// TIA Portal V17 export
// export: Created 2026-04-12T10:31:24.245585Z, ExportSetting WithDefaults, DisplayName Totally Integrated Automation Portal, DisplayVersion V17 Update 4, DisplayName TIA Portal Openness, DisplayVersion V17 Update 4, DisplayName TIA Portal Version Control Interface, DisplayVersion V17, DisplayName SINAMICS Startdrive Advanced, DisplayVersion V17, DisplayName SINAMICS Startdrive G130, G150, S120, S150, SINAMICS MV, S210, DisplayVersion V17, DisplayName SINAMICS Startdrive G110M, G120, G120C, G120D, G120P, G115D, DisplayVersion V17, DisplayName STEP 7 Professional, DisplayVersion V17 Update 4, DisplayName STEP 7 Safety, DisplayVersion V17, DisplayName WinCC Advanced, DisplayVersion V17 Update 4
FUNCTION "烧嘴控制块" : Void   // FC4, LAD
{ S7_Optimized_Access := 'TRUE' }
VERSION : 0.1
// stored: AutoNumber true, IsIECCheckEnabled false, SetENOAutomatically false, UDAEnableTagReadback false
   VAR_TEMP   // added for the SCL form of the ladder/FBD networks
      _w1 : Bool;
      _w2 : Bool;
   END_VAR
BEGIN

REGION Network 1: 1#烧嘴控制
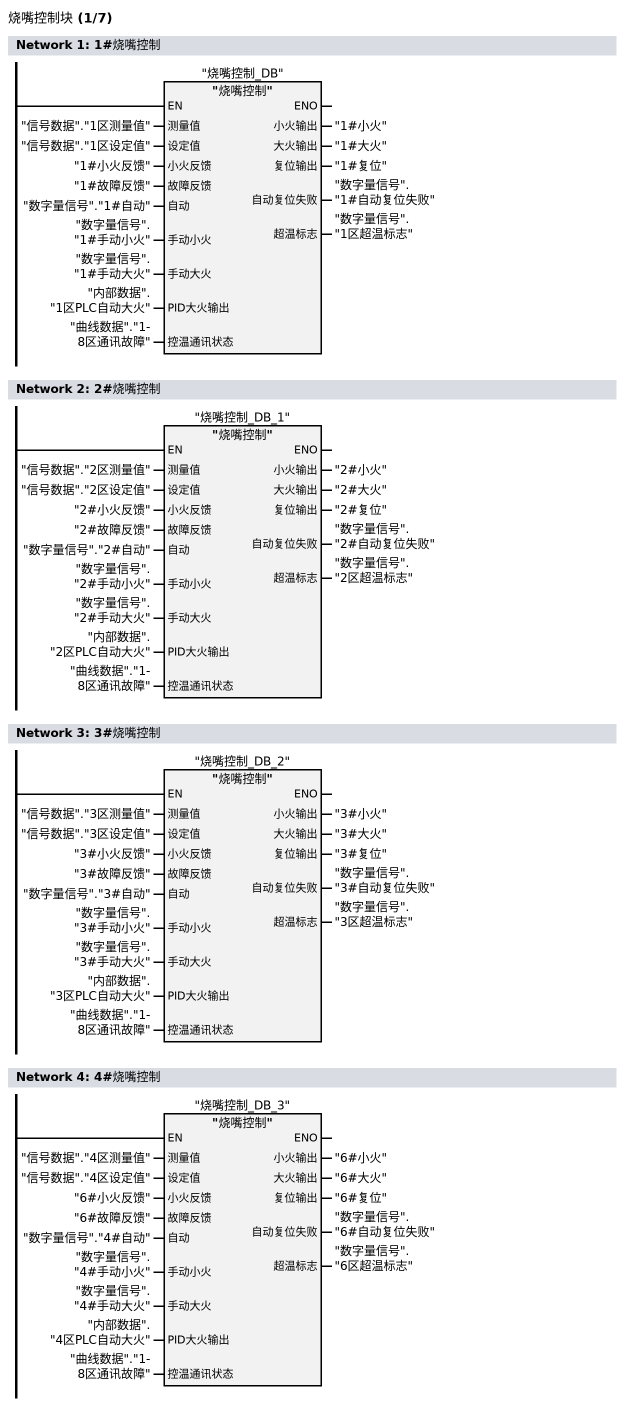
   RUNG wire#powerrail
      "烧嘴控制_DB"(测量值 := "信号数据"."1区测量值", 设定值 := "信号数据"."1区设定值", 小火反馈 := "1#小火反馈", 故障反馈 := "1#故障反馈", 自动 := "数字量信号"."1#自动", 手动小火 := "数字量信号"."1#手动小火", 手动大火 := "数字量信号"."1#手动大火", PID大火输出 := "内部数据"."1区PLC自动大火", 控温通讯状态 := "曲线数据"."1-8区通讯故障", 小火输出 => "1#小火", 大火输出 => "1#大火", 复位输出 => "1#复位", 自动复位失败 => "数字量信号"."1#自动复位失败", 超温标志 => "数字量信号"."1区超温标志")
   END_RUNG
   // the same network as SCL:
   "烧嘴控制_DB"(测量值 := "信号数据"."1区测量值",   // "烧嘴控制"
             设定值 := "信号数据"."1区设定值",
             小火反馈 := "1#小火反馈",
             故障反馈 := "1#故障反馈",
             自动 := "数字量信号"."1#自动",
             手动小火 := "数字量信号"."1#手动小火",
             手动大火 := "数字量信号"."1#手动大火",
             PID大火输出 := "内部数据"."1区PLC自动大火",
             控温通讯状态 := "曲线数据"."1-8区通讯故障",
             小火输出 => "1#小火",
             大火输出 => "1#大火",
             复位输出 => "1#复位",
             自动复位失败 => "数字量信号"."1#自动复位失败",
             超温标志 => "数字量信号"."1区超温标志");
END_REGION

REGION Network 2: 2#烧嘴控制
   RUNG wire#powerrail
      "烧嘴控制_DB_1"(测量值 := "信号数据"."2区测量值", 设定值 := "信号数据"."2区设定值", 小火反馈 := "2#小火反馈", 故障反馈 := "2#故障反馈", 自动 := "数字量信号"."2#自动", 手动小火 := "数字量信号"."2#手动小火", 手动大火 := "数字量信号"."2#手动大火", PID大火输出 := "内部数据"."2区PLC自动大火", 控温通讯状态 := "曲线数据"."1-8区通讯故障", 小火输出 => "2#小火", 大火输出 => "2#大火", 复位输出 => "2#复位", 自动复位失败 => "数字量信号"."2#自动复位失败", 超温标志 => "数字量信号"."2区超温标志")
   END_RUNG
   // the same network as SCL:
   "烧嘴控制_DB_1"(测量值 := "信号数据"."2区测量值",   // "烧嘴控制"
               设定值 := "信号数据"."2区设定值",
               小火反馈 := "2#小火反馈",
               故障反馈 := "2#故障反馈",
               自动 := "数字量信号"."2#自动",
               手动小火 := "数字量信号"."2#手动小火",
               手动大火 := "数字量信号"."2#手动大火",
               PID大火输出 := "内部数据"."2区PLC自动大火",
               控温通讯状态 := "曲线数据"."1-8区通讯故障",
               小火输出 => "2#小火",
               大火输出 => "2#大火",
               复位输出 => "2#复位",
               自动复位失败 => "数字量信号"."2#自动复位失败",
               超温标志 => "数字量信号"."2区超温标志");
END_REGION

REGION Network 3: 3#烧嘴控制
   RUNG wire#powerrail
      "烧嘴控制_DB_2"(测量值 := "信号数据"."3区测量值", 设定值 := "信号数据"."3区设定值", 小火反馈 := "3#小火反馈", 故障反馈 := "3#故障反馈", 自动 := "数字量信号"."3#自动", 手动小火 := "数字量信号"."3#手动小火", 手动大火 := "数字量信号"."3#手动大火", PID大火输出 := "内部数据"."3区PLC自动大火", 控温通讯状态 := "曲线数据"."1-8区通讯故障", 小火输出 => "3#小火", 大火输出 => "3#大火", 复位输出 => "3#复位", 自动复位失败 => "数字量信号"."3#自动复位失败", 超温标志 => "数字量信号"."3区超温标志")
   END_RUNG
   // the same network as SCL:
   "烧嘴控制_DB_2"(测量值 := "信号数据"."3区测量值",   // "烧嘴控制"
               设定值 := "信号数据"."3区设定值",
               小火反馈 := "3#小火反馈",
               故障反馈 := "3#故障反馈",
               自动 := "数字量信号"."3#自动",
               手动小火 := "数字量信号"."3#手动小火",
               手动大火 := "数字量信号"."3#手动大火",
               PID大火输出 := "内部数据"."3区PLC自动大火",
               控温通讯状态 := "曲线数据"."1-8区通讯故障",
               小火输出 => "3#小火",
               大火输出 => "3#大火",
               复位输出 => "3#复位",
               自动复位失败 => "数字量信号"."3#自动复位失败",
               超温标志 => "数字量信号"."3区超温标志");
END_REGION

REGION Network 4: 4#烧嘴控制
   RUNG wire#powerrail
      "烧嘴控制_DB_3"(测量值 := "信号数据"."4区测量值", 设定值 := "信号数据"."4区设定值", 小火反馈 := "6#小火反馈", 故障反馈 := "6#故障反馈", 自动 := "数字量信号"."4#自动", 手动小火 := "数字量信号"."4#手动小火", 手动大火 := "数字量信号"."4#手动大火", PID大火输出 := "内部数据"."4区PLC自动大火", 控温通讯状态 := "曲线数据"."1-8区通讯故障", 小火输出 => "6#小火", 大火输出 => "6#大火", 复位输出 => "6#复位", 自动复位失败 => "数字量信号"."6#自动复位失败", 超温标志 => "数字量信号"."6区超温标志")
   END_RUNG
   // the same network as SCL:
   "烧嘴控制_DB_3"(测量值 := "信号数据"."4区测量值",   // "烧嘴控制"
               设定值 := "信号数据"."4区设定值",
               小火反馈 := "6#小火反馈",
               故障反馈 := "6#故障反馈",
               自动 := "数字量信号"."4#自动",
               手动小火 := "数字量信号"."4#手动小火",
               手动大火 := "数字量信号"."4#手动大火",
               PID大火输出 := "内部数据"."4区PLC自动大火",
               控温通讯状态 := "曲线数据"."1-8区通讯故障",
               小火输出 => "6#小火",
               大火输出 => "6#大火",
               复位输出 => "6#复位",
               自动复位失败 => "数字量信号"."6#自动复位失败",
               超温标志 => "数字量信号"."6区超温标志");
END_REGION

REGION Network 5: 5#烧嘴控制
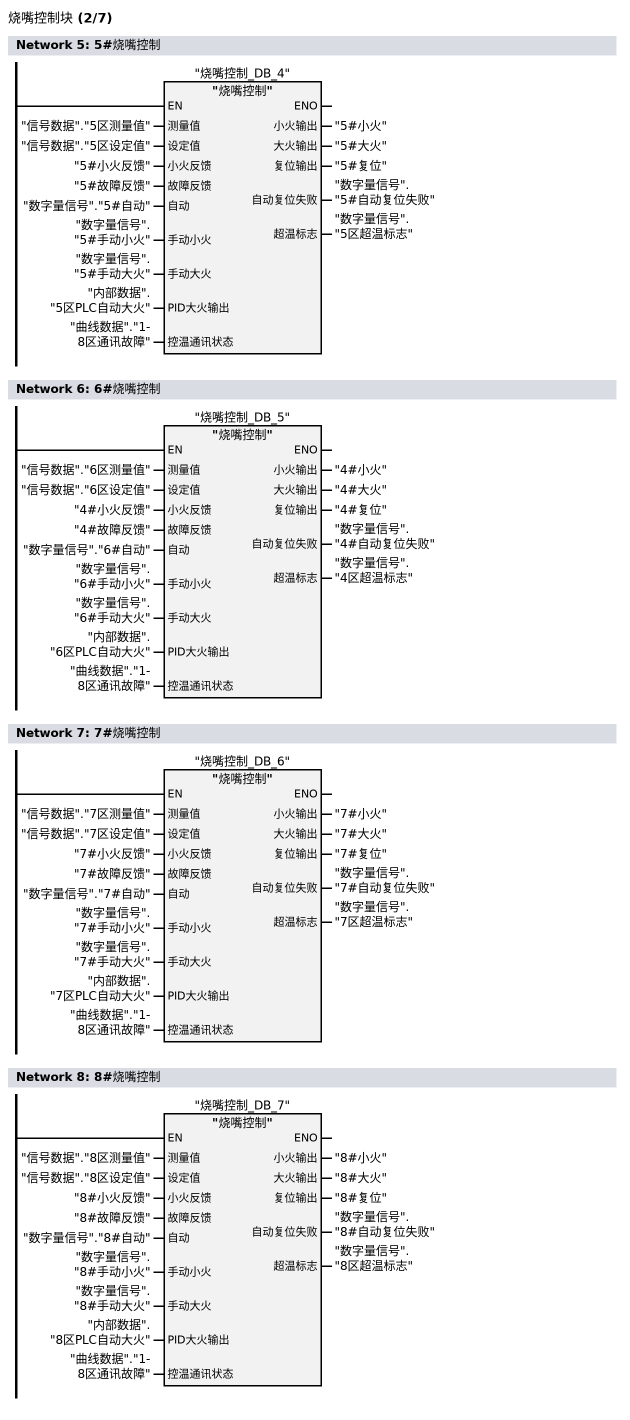
   RUNG wire#powerrail
      "烧嘴控制_DB_4"(测量值 := "信号数据"."5区测量值", 设定值 := "信号数据"."5区设定值", 小火反馈 := "5#小火反馈", 故障反馈 := "5#故障反馈", 自动 := "数字量信号"."5#自动", 手动小火 := "数字量信号"."5#手动小火", 手动大火 := "数字量信号"."5#手动大火", PID大火输出 := "内部数据"."5区PLC自动大火", 控温通讯状态 := "曲线数据"."1-8区通讯故障", 小火输出 => "5#小火", 大火输出 => "5#大火", 复位输出 => "5#复位", 自动复位失败 => "数字量信号"."5#自动复位失败", 超温标志 => "数字量信号"."5区超温标志")
   END_RUNG
   // the same network as SCL:
   "烧嘴控制_DB_4"(测量值 := "信号数据"."5区测量值",   // "烧嘴控制"
               设定值 := "信号数据"."5区设定值",
               小火反馈 := "5#小火反馈",
               故障反馈 := "5#故障反馈",
               自动 := "数字量信号"."5#自动",
               手动小火 := "数字量信号"."5#手动小火",
               手动大火 := "数字量信号"."5#手动大火",
               PID大火输出 := "内部数据"."5区PLC自动大火",
               控温通讯状态 := "曲线数据"."1-8区通讯故障",
               小火输出 => "5#小火",
               大火输出 => "5#大火",
               复位输出 => "5#复位",
               自动复位失败 => "数字量信号"."5#自动复位失败",
               超温标志 => "数字量信号"."5区超温标志");
END_REGION

REGION Network 6: 6#烧嘴控制
   RUNG wire#powerrail
      "烧嘴控制_DB_5"(测量值 := "信号数据"."6区测量值", 设定值 := "信号数据"."6区设定值", 小火反馈 := "4#小火反馈", 故障反馈 := "4#故障反馈", 自动 := "数字量信号"."6#自动", 手动小火 := "数字量信号"."6#手动小火", 手动大火 := "数字量信号"."6#手动大火", PID大火输出 := "内部数据"."6区PLC自动大火", 控温通讯状态 := "曲线数据"."1-8区通讯故障", 小火输出 => "4#小火", 大火输出 => "4#大火", 复位输出 => "4#复位", 自动复位失败 => "数字量信号"."4#自动复位失败", 超温标志 => "数字量信号"."4区超温标志")
   END_RUNG
   // the same network as SCL:
   "烧嘴控制_DB_5"(测量值 := "信号数据"."6区测量值",   // "烧嘴控制"
               设定值 := "信号数据"."6区设定值",
               小火反馈 := "4#小火反馈",
               故障反馈 := "4#故障反馈",
               自动 := "数字量信号"."6#自动",
               手动小火 := "数字量信号"."6#手动小火",
               手动大火 := "数字量信号"."6#手动大火",
               PID大火输出 := "内部数据"."6区PLC自动大火",
               控温通讯状态 := "曲线数据"."1-8区通讯故障",
               小火输出 => "4#小火",
               大火输出 => "4#大火",
               复位输出 => "4#复位",
               自动复位失败 => "数字量信号"."4#自动复位失败",
               超温标志 => "数字量信号"."4区超温标志");
END_REGION

REGION Network 7: 7#烧嘴控制
   RUNG wire#powerrail
      "烧嘴控制_DB_6"(测量值 := "信号数据"."7区测量值", 设定值 := "信号数据"."7区设定值", 小火反馈 := "7#小火反馈", 故障反馈 := "7#故障反馈", 自动 := "数字量信号"."7#自动", 手动小火 := "数字量信号"."7#手动小火", 手动大火 := "数字量信号"."7#手动大火", PID大火输出 := "内部数据"."7区PLC自动大火", 控温通讯状态 := "曲线数据"."1-8区通讯故障", 小火输出 => "7#小火", 大火输出 => "7#大火", 复位输出 => "7#复位", 自动复位失败 => "数字量信号"."7#自动复位失败", 超温标志 => "数字量信号"."7区超温标志")
   END_RUNG
   // the same network as SCL:
   "烧嘴控制_DB_6"(测量值 := "信号数据"."7区测量值",   // "烧嘴控制"
               设定值 := "信号数据"."7区设定值",
               小火反馈 := "7#小火反馈",
               故障反馈 := "7#故障反馈",
               自动 := "数字量信号"."7#自动",
               手动小火 := "数字量信号"."7#手动小火",
               手动大火 := "数字量信号"."7#手动大火",
               PID大火输出 := "内部数据"."7区PLC自动大火",
               控温通讯状态 := "曲线数据"."1-8区通讯故障",
               小火输出 => "7#小火",
               大火输出 => "7#大火",
               复位输出 => "7#复位",
               自动复位失败 => "数字量信号"."7#自动复位失败",
               超温标志 => "数字量信号"."7区超温标志");
END_REGION

REGION Network 8: 8#烧嘴控制
   RUNG wire#powerrail
      "烧嘴控制_DB_7"(测量值 := "信号数据"."8区测量值", 设定值 := "信号数据"."8区设定值", 小火反馈 := "8#小火反馈", 故障反馈 := "8#故障反馈", 自动 := "数字量信号"."8#自动", 手动小火 := "数字量信号"."8#手动小火", 手动大火 := "数字量信号"."8#手动大火", PID大火输出 := "内部数据"."8区PLC自动大火", 控温通讯状态 := "曲线数据"."1-8区通讯故障", 小火输出 => "8#小火", 大火输出 => "8#大火", 复位输出 => "8#复位", 自动复位失败 => "数字量信号"."8#自动复位失败", 超温标志 => "数字量信号"."8区超温标志")
   END_RUNG
   // the same network as SCL:
   "烧嘴控制_DB_7"(测量值 := "信号数据"."8区测量值",   // "烧嘴控制"
               设定值 := "信号数据"."8区设定值",
               小火反馈 := "8#小火反馈",
               故障反馈 := "8#故障反馈",
               自动 := "数字量信号"."8#自动",
               手动小火 := "数字量信号"."8#手动小火",
               手动大火 := "数字量信号"."8#手动大火",
               PID大火输出 := "内部数据"."8区PLC自动大火",
               控温通讯状态 := "曲线数据"."1-8区通讯故障",
               小火输出 => "8#小火",
               大火输出 => "8#大火",
               复位输出 => "8#复位",
               自动复位失败 => "数字量信号"."8#自动复位失败",
               超温标志 => "数字量信号"."8区超温标志");
END_REGION

REGION Network 9: 9#烧嘴控制
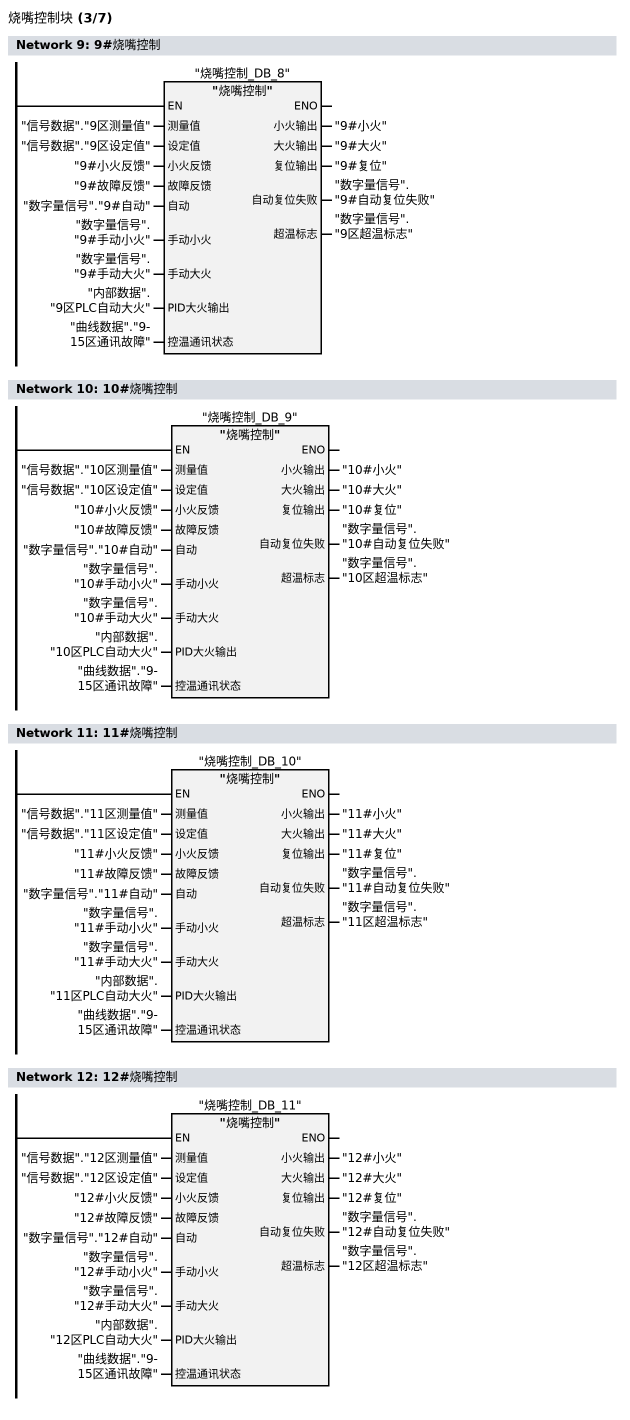
   RUNG wire#powerrail
      "烧嘴控制_DB_8"(测量值 := "信号数据"."9区测量值", 设定值 := "信号数据"."9区设定值", 小火反馈 := "9#小火反馈", 故障反馈 := "9#故障反馈", 自动 := "数字量信号"."9#自动", 手动小火 := "数字量信号"."9#手动小火", 手动大火 := "数字量信号"."9#手动大火", PID大火输出 := "内部数据"."9区PLC自动大火", 控温通讯状态 := "曲线数据"."9-15区通讯故障", 小火输出 => "9#小火", 大火输出 => "9#大火", 复位输出 => "9#复位", 自动复位失败 => "数字量信号"."9#自动复位失败", 超温标志 => "数字量信号"."9区超温标志")
   END_RUNG
   // the same network as SCL:
   "烧嘴控制_DB_8"(测量值 := "信号数据"."9区测量值",   // "烧嘴控制"
               设定值 := "信号数据"."9区设定值",
               小火反馈 := "9#小火反馈",
               故障反馈 := "9#故障反馈",
               自动 := "数字量信号"."9#自动",
               手动小火 := "数字量信号"."9#手动小火",
               手动大火 := "数字量信号"."9#手动大火",
               PID大火输出 := "内部数据"."9区PLC自动大火",
               控温通讯状态 := "曲线数据"."9-15区通讯故障",
               小火输出 => "9#小火",
               大火输出 => "9#大火",
               复位输出 => "9#复位",
               自动复位失败 => "数字量信号"."9#自动复位失败",
               超温标志 => "数字量信号"."9区超温标志");
END_REGION

REGION Network 10: 10#烧嘴控制
   RUNG wire#powerrail
      "烧嘴控制_DB_9"(测量值 := "信号数据"."10区测量值", 设定值 := "信号数据"."10区设定值", 小火反馈 := "10#小火反馈", 故障反馈 := "10#故障反馈", 自动 := "数字量信号"."10#自动", 手动小火 := "数字量信号"."10#手动小火", 手动大火 := "数字量信号"."10#手动大火", PID大火输出 := "内部数据"."10区PLC自动大火", 控温通讯状态 := "曲线数据"."9-15区通讯故障", 小火输出 => "10#小火", 大火输出 => "10#大火", 复位输出 => "10#复位", 自动复位失败 => "数字量信号"."10#自动复位失败", 超温标志 => "数字量信号"."10区超温标志")
   END_RUNG
   // the same network as SCL:
   "烧嘴控制_DB_9"(测量值 := "信号数据"."10区测量值",   // "烧嘴控制"
               设定值 := "信号数据"."10区设定值",
               小火反馈 := "10#小火反馈",
               故障反馈 := "10#故障反馈",
               自动 := "数字量信号"."10#自动",
               手动小火 := "数字量信号"."10#手动小火",
               手动大火 := "数字量信号"."10#手动大火",
               PID大火输出 := "内部数据"."10区PLC自动大火",
               控温通讯状态 := "曲线数据"."9-15区通讯故障",
               小火输出 => "10#小火",
               大火输出 => "10#大火",
               复位输出 => "10#复位",
               自动复位失败 => "数字量信号"."10#自动复位失败",
               超温标志 => "数字量信号"."10区超温标志");
END_REGION

REGION Network 11: 11#烧嘴控制
   RUNG wire#powerrail
      "烧嘴控制_DB_10"(测量值 := "信号数据"."11区测量值", 设定值 := "信号数据"."11区设定值", 小火反馈 := "11#小火反馈", 故障反馈 := "11#故障反馈", 自动 := "数字量信号"."11#自动", 手动小火 := "数字量信号"."11#手动小火", 手动大火 := "数字量信号"."11#手动大火", PID大火输出 := "内部数据"."11区PLC自动大火", 控温通讯状态 := "曲线数据"."9-15区通讯故障", 小火输出 => "11#小火", 大火输出 => "11#大火", 复位输出 => "11#复位", 自动复位失败 => "数字量信号"."11#自动复位失败", 超温标志 => "数字量信号"."11区超温标志")
   END_RUNG
   // the same network as SCL:
   "烧嘴控制_DB_10"(测量值 := "信号数据"."11区测量值",   // "烧嘴控制"
                设定值 := "信号数据"."11区设定值",
                小火反馈 := "11#小火反馈",
                故障反馈 := "11#故障反馈",
                自动 := "数字量信号"."11#自动",
                手动小火 := "数字量信号"."11#手动小火",
                手动大火 := "数字量信号"."11#手动大火",
                PID大火输出 := "内部数据"."11区PLC自动大火",
                控温通讯状态 := "曲线数据"."9-15区通讯故障",
                小火输出 => "11#小火",
                大火输出 => "11#大火",
                复位输出 => "11#复位",
                自动复位失败 => "数字量信号"."11#自动复位失败",
                超温标志 => "数字量信号"."11区超温标志");
END_REGION

REGION Network 12: 12#烧嘴控制
   RUNG wire#powerrail
      "烧嘴控制_DB_11"(测量值 := "信号数据"."12区测量值", 设定值 := "信号数据"."12区设定值", 小火反馈 := "12#小火反馈", 故障反馈 := "12#故障反馈", 自动 := "数字量信号"."12#自动", 手动小火 := "数字量信号"."12#手动小火", 手动大火 := "数字量信号"."12#手动大火", PID大火输出 := "内部数据"."12区PLC自动大火", 控温通讯状态 := "曲线数据"."9-15区通讯故障", 小火输出 => "12#小火", 大火输出 => "12#大火", 复位输出 => "12#复位", 自动复位失败 => "数字量信号"."12#自动复位失败", 超温标志 => "数字量信号"."12区超温标志")
   END_RUNG
   // the same network as SCL:
   "烧嘴控制_DB_11"(测量值 := "信号数据"."12区测量值",   // "烧嘴控制"
                设定值 := "信号数据"."12区设定值",
                小火反馈 := "12#小火反馈",
                故障反馈 := "12#故障反馈",
                自动 := "数字量信号"."12#自动",
                手动小火 := "数字量信号"."12#手动小火",
                手动大火 := "数字量信号"."12#手动大火",
                PID大火输出 := "内部数据"."12区PLC自动大火",
                控温通讯状态 := "曲线数据"."9-15区通讯故障",
                小火输出 => "12#小火",
                大火输出 => "12#大火",
                复位输出 => "12#复位",
                自动复位失败 => "数字量信号"."12#自动复位失败",
                超温标志 => "数字量信号"."12区超温标志");
END_REGION

REGION Network 13: 13#烧嘴控制
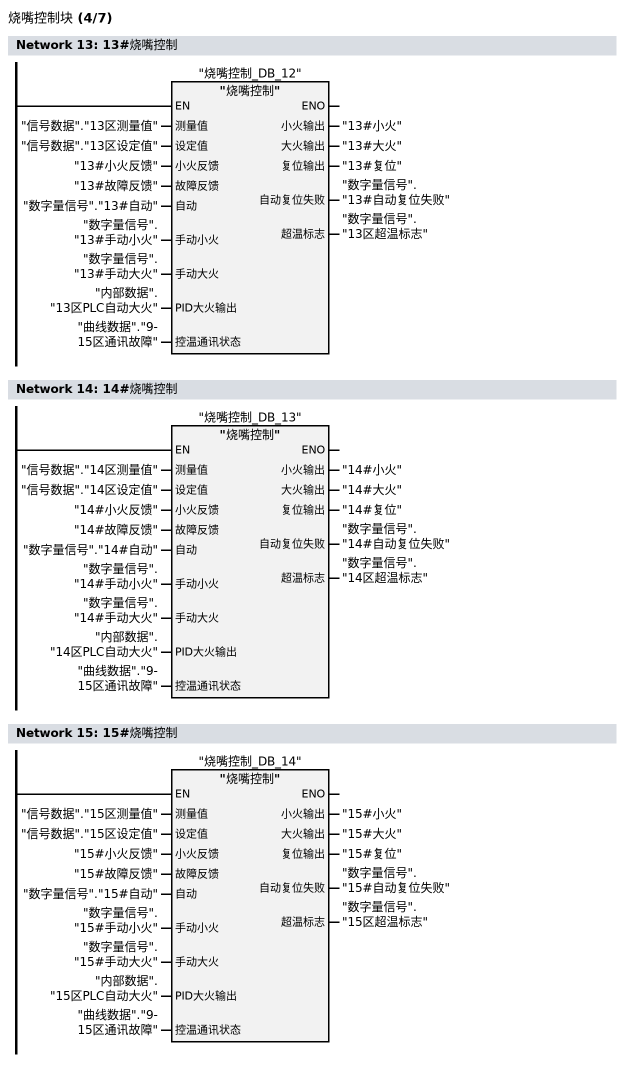
   RUNG wire#powerrail
      "烧嘴控制_DB_12"(测量值 := "信号数据"."13区测量值", 设定值 := "信号数据"."13区设定值", 小火反馈 := "13#小火反馈", 故障反馈 := "13#故障反馈", 自动 := "数字量信号"."13#自动", 手动小火 := "数字量信号"."13#手动小火", 手动大火 := "数字量信号"."13#手动大火", PID大火输出 := "内部数据"."13区PLC自动大火", 控温通讯状态 := "曲线数据"."9-15区通讯故障", 小火输出 => "13#小火", 大火输出 => "13#大火", 复位输出 => "13#复位", 自动复位失败 => "数字量信号"."13#自动复位失败", 超温标志 => "数字量信号"."13区超温标志")
   END_RUNG
   // the same network as SCL:
   "烧嘴控制_DB_12"(测量值 := "信号数据"."13区测量值",   // "烧嘴控制"
                设定值 := "信号数据"."13区设定值",
                小火反馈 := "13#小火反馈",
                故障反馈 := "13#故障反馈",
                自动 := "数字量信号"."13#自动",
                手动小火 := "数字量信号"."13#手动小火",
                手动大火 := "数字量信号"."13#手动大火",
                PID大火输出 := "内部数据"."13区PLC自动大火",
                控温通讯状态 := "曲线数据"."9-15区通讯故障",
                小火输出 => "13#小火",
                大火输出 => "13#大火",
                复位输出 => "13#复位",
                自动复位失败 => "数字量信号"."13#自动复位失败",
                超温标志 => "数字量信号"."13区超温标志");
END_REGION

REGION Network 14: 14#烧嘴控制
   RUNG wire#powerrail
      "烧嘴控制_DB_13"(测量值 := "信号数据"."14区测量值", 设定值 := "信号数据"."14区设定值", 小火反馈 := "14#小火反馈", 故障反馈 := "14#故障反馈", 自动 := "数字量信号"."14#自动", 手动小火 := "数字量信号"."14#手动小火", 手动大火 := "数字量信号"."14#手动大火", PID大火输出 := "内部数据"."14区PLC自动大火", 控温通讯状态 := "曲线数据"."9-15区通讯故障", 小火输出 => "14#小火", 大火输出 => "14#大火", 复位输出 => "14#复位", 自动复位失败 => "数字量信号"."14#自动复位失败", 超温标志 => "数字量信号"."14区超温标志")
   END_RUNG
   // the same network as SCL:
   "烧嘴控制_DB_13"(测量值 := "信号数据"."14区测量值",   // "烧嘴控制"
                设定值 := "信号数据"."14区设定值",
                小火反馈 := "14#小火反馈",
                故障反馈 := "14#故障反馈",
                自动 := "数字量信号"."14#自动",
                手动小火 := "数字量信号"."14#手动小火",
                手动大火 := "数字量信号"."14#手动大火",
                PID大火输出 := "内部数据"."14区PLC自动大火",
                控温通讯状态 := "曲线数据"."9-15区通讯故障",
                小火输出 => "14#小火",
                大火输出 => "14#大火",
                复位输出 => "14#复位",
                自动复位失败 => "数字量信号"."14#自动复位失败",
                超温标志 => "数字量信号"."14区超温标志");
END_REGION

REGION Network 15: 15#烧嘴控制
   RUNG wire#powerrail
      "烧嘴控制_DB_14"(测量值 := "信号数据"."15区测量值", 设定值 := "信号数据"."15区设定值", 小火反馈 := "15#小火反馈", 故障反馈 := "15#故障反馈", 自动 := "数字量信号"."15#自动", 手动小火 := "数字量信号"."15#手动小火", 手动大火 := "数字量信号"."15#手动大火", PID大火输出 := "内部数据"."15区PLC自动大火", 控温通讯状态 := "曲线数据"."9-15区通讯故障", 小火输出 => "15#小火", 大火输出 => "15#大火", 复位输出 => "15#复位", 自动复位失败 => "数字量信号"."15#自动复位失败", 超温标志 => "数字量信号"."15区超温标志")
   END_RUNG
   // the same network as SCL:
   "烧嘴控制_DB_14"(测量值 := "信号数据"."15区测量值",   // "烧嘴控制"
                设定值 := "信号数据"."15区设定值",
                小火反馈 := "15#小火反馈",
                故障反馈 := "15#故障反馈",
                自动 := "数字量信号"."15#自动",
                手动小火 := "数字量信号"."15#手动小火",
                手动大火 := "数字量信号"."15#手动大火",
                PID大火输出 := "内部数据"."15区PLC自动大火",
                控温通讯状态 := "曲线数据"."9-15区通讯故障",
                小火输出 => "15#小火",
                大火输出 => "15#大火",
                复位输出 => "15#复位",
                自动复位失败 => "数字量信号"."15#自动复位失败",
                超温标志 => "数字量信号"."15区超温标志");
END_REGION

REGION Network 16: 烧嘴复位失败标志
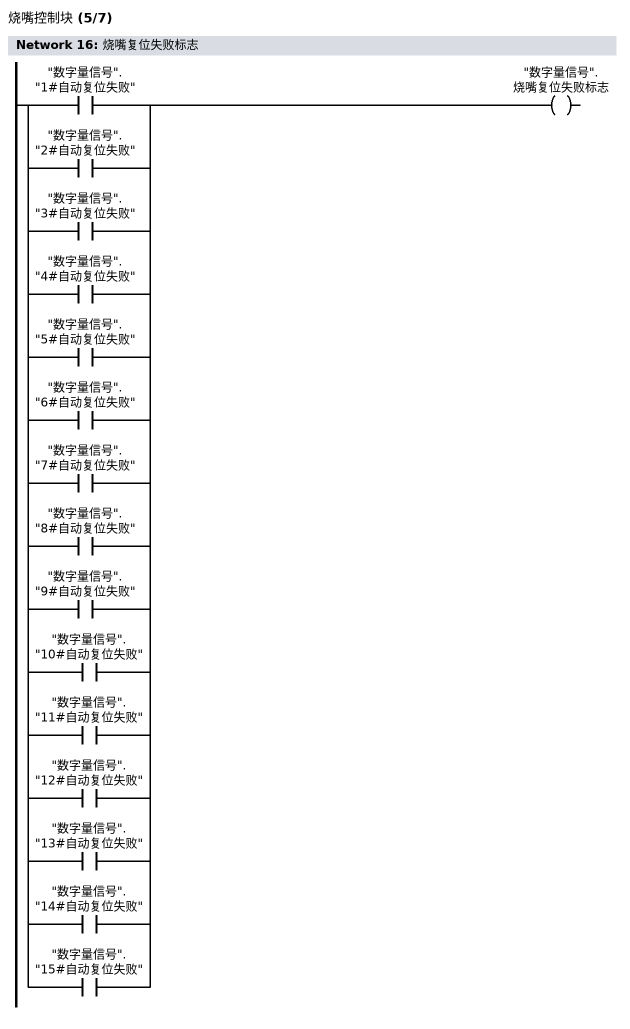
   RUNG wire#powerrail
      Contact( "数字量信号"."1#自动复位失败" )
      wire#w1
      Coil( "数字量信号".烧嘴复位失败标志 )
   END_RUNG
   RUNG wire#powerrail
      Contact( "数字量信号"."2#自动复位失败" )
   END_RUNG wire#w1
   RUNG wire#powerrail
      Contact( "数字量信号"."3#自动复位失败" )
   END_RUNG wire#w1
   RUNG wire#powerrail
      Contact( "数字量信号"."4#自动复位失败" )
   END_RUNG wire#w1
   RUNG wire#powerrail
      Contact( "数字量信号"."5#自动复位失败" )
   END_RUNG wire#w1
   RUNG wire#powerrail
      Contact( "数字量信号"."6#自动复位失败" )
   END_RUNG wire#w1
   RUNG wire#powerrail
      Contact( "数字量信号"."7#自动复位失败" )
   END_RUNG wire#w1
   RUNG wire#powerrail
      Contact( "数字量信号"."8#自动复位失败" )
   END_RUNG wire#w1
   RUNG wire#powerrail
      Contact( "数字量信号"."9#自动复位失败" )
   END_RUNG wire#w1
   RUNG wire#powerrail
      Contact( "数字量信号"."10#自动复位失败" )
   END_RUNG wire#w1
   RUNG wire#powerrail
      Contact( "数字量信号"."11#自动复位失败" )
   END_RUNG wire#w1
   RUNG wire#powerrail
      Contact( "数字量信号"."12#自动复位失败" )
   END_RUNG wire#w1
   RUNG wire#powerrail
      Contact( "数字量信号"."13#自动复位失败" )
   END_RUNG wire#w1
   RUNG wire#powerrail
      Contact( "数字量信号"."14#自动复位失败" )
   END_RUNG wire#w1
   RUNG wire#powerrail
      Contact( "数字量信号"."15#自动复位失败" )
   END_RUNG wire#w1
   // the same network as SCL:
   "数字量信号".烧嘴复位失败标志 := "数字量信号"."1#自动复位失败" OR "数字量信号"."2#自动复位失败" OR "数字量信号"."3#自动复位失败" OR "数字量信号"."4#自动复位失败" OR "数字量信号"."5#自动复位失败" OR "数字量信号"."6#自动复位失败" OR "数字量信号"."7#自动复位失败" OR "数字量信号"."8#自动复位失败" OR "数字量信号"."9#自动复位失败" OR "数字量信号"."10#自动复位失败" OR "数字量信号"."11#自动复位失败" OR "数字量信号"."12#自动复位失败" OR "数字量信号"."13#自动复位失败" OR "数字量信号"."14#自动复位失败" OR "数字量信号"."15#自动复位失败";
END_REGION

REGION Network 17: 烧嘴报警
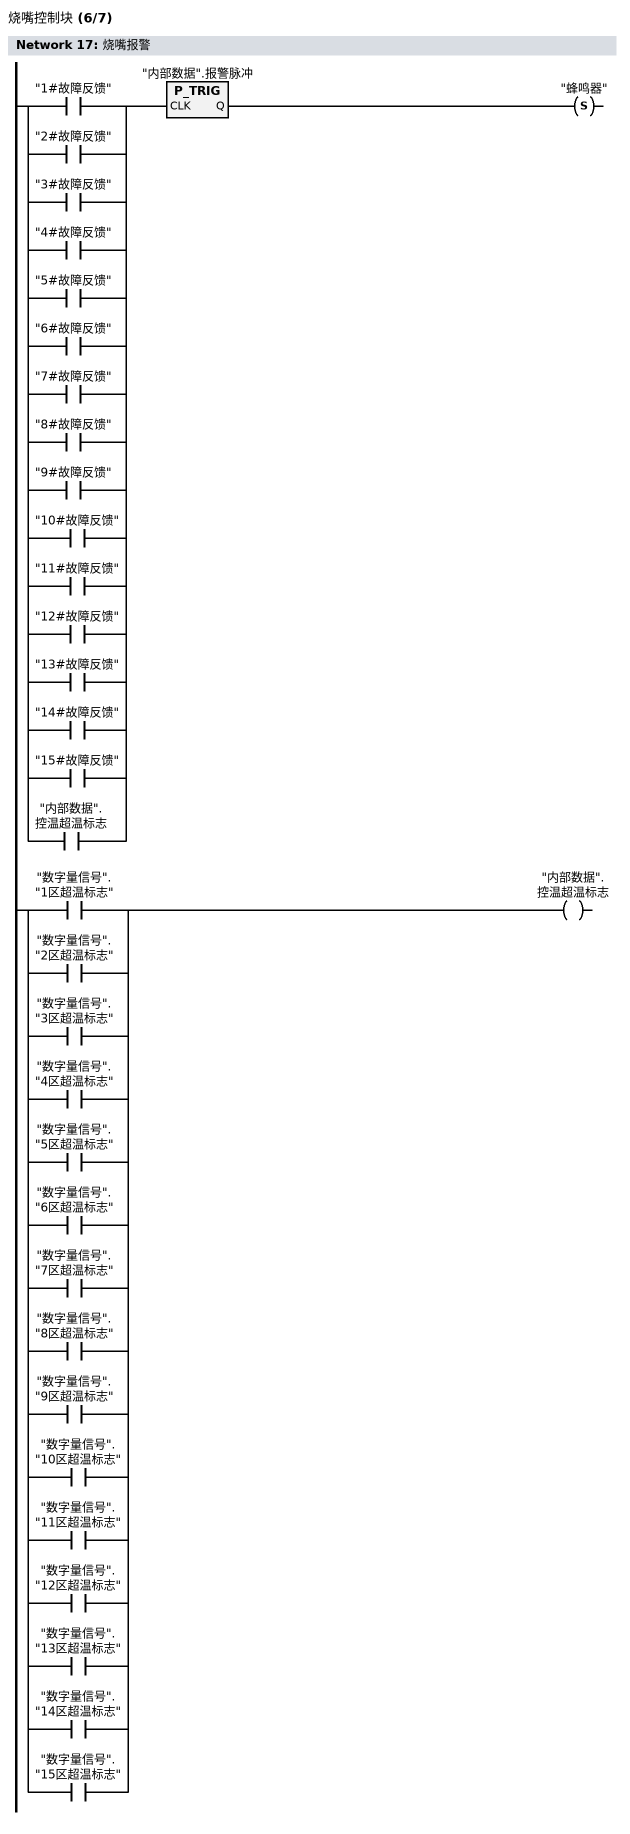
   RUNG wire#powerrail
      Contact( "1#故障反馈" )
      wire#w1
      P_Trig( "内部数据".报警脉冲 )
      S_Coil( "蜂鸣器" )
   END_RUNG
   RUNG wire#powerrail
      Contact( "2#故障反馈" )
   END_RUNG wire#w1
   RUNG wire#powerrail
      Contact( "3#故障反馈" )
   END_RUNG wire#w1
   RUNG wire#powerrail
      Contact( "4#故障反馈" )
   END_RUNG wire#w1
   RUNG wire#powerrail
      Contact( "5#故障反馈" )
   END_RUNG wire#w1
   RUNG wire#powerrail
      Contact( "6#故障反馈" )
   END_RUNG wire#w1
   RUNG wire#powerrail
      Contact( "7#故障反馈" )
   END_RUNG wire#w1
   RUNG wire#powerrail
      Contact( "8#故障反馈" )
   END_RUNG wire#w1
   RUNG wire#powerrail
      Contact( "9#故障反馈" )
   END_RUNG wire#w1
   RUNG wire#powerrail
      Contact( "10#故障反馈" )
   END_RUNG wire#w1
   RUNG wire#powerrail
      Contact( "11#故障反馈" )
   END_RUNG wire#w1
   RUNG wire#powerrail
      Contact( "12#故障反馈" )
   END_RUNG wire#w1
   RUNG wire#powerrail
      Contact( "13#故障反馈" )
   END_RUNG wire#w1
   RUNG wire#powerrail
      Contact( "14#故障反馈" )
   END_RUNG wire#w1
   RUNG wire#powerrail
      Contact( "15#故障反馈" )
   END_RUNG wire#w1
   RUNG wire#powerrail
      Contact( "内部数据".控温超温标志 )
   END_RUNG wire#w1
   RUNG wire#powerrail
      Contact( "数字量信号"."1区超温标志" )
      wire#w2
      Coil( "内部数据".控温超温标志 )
   END_RUNG
   RUNG wire#powerrail
      Contact( "数字量信号"."2区超温标志" )
   END_RUNG wire#w2
   RUNG wire#powerrail
      Contact( "数字量信号"."3区超温标志" )
   END_RUNG wire#w2
   RUNG wire#powerrail
      Contact( "数字量信号"."4区超温标志" )
   END_RUNG wire#w2
   RUNG wire#powerrail
      Contact( "数字量信号"."5区超温标志" )
   END_RUNG wire#w2
   RUNG wire#powerrail
      Contact( "数字量信号"."6区超温标志" )
   END_RUNG wire#w2
   RUNG wire#powerrail
      Contact( "数字量信号"."7区超温标志" )
   END_RUNG wire#w2
   RUNG wire#powerrail
      Contact( "数字量信号"."8区超温标志" )
   END_RUNG wire#w2
   RUNG wire#powerrail
      Contact( "数字量信号"."9区超温标志" )
   END_RUNG wire#w2
   RUNG wire#powerrail
      Contact( "数字量信号"."10区超温标志" )
   END_RUNG wire#w2
   RUNG wire#powerrail
      Contact( "数字量信号"."11区超温标志" )
   END_RUNG wire#w2
   RUNG wire#powerrail
      Contact( "数字量信号"."12区超温标志" )
   END_RUNG wire#w2
   RUNG wire#powerrail
      Contact( "数字量信号"."13区超温标志" )
   END_RUNG wire#w2
   RUNG wire#powerrail
      Contact( "数字量信号"."14区超温标志" )
   END_RUNG wire#w2
   RUNG wire#powerrail
      Contact( "数字量信号"."15区超温标志" )
   END_RUNG wire#w2
   // the same network as SCL:
   #_w1 := "1#故障反馈" OR "2#故障反馈" OR "3#故障反馈" OR "4#故障反馈" OR "5#故障反馈" OR "6#故障反馈" OR "7#故障反馈" OR "8#故障反馈" OR "9#故障反馈" OR "10#故障反馈" OR "11#故障反馈" OR "12#故障反馈" OR "13#故障反馈" OR "14#故障反馈" OR "15#故障反馈" OR "内部数据".控温超温标志;
   #_w2 := #_w1 AND NOT "内部数据".报警脉冲;   // rising edge
   "内部数据".报警脉冲 := #_w1;
   IF #_w2 THEN "蜂鸣器" := TRUE; END_IF;
   "内部数据".控温超温标志 := "数字量信号"."1区超温标志" OR "数字量信号"."2区超温标志" OR "数字量信号"."3区超温标志" OR "数字量信号"."4区超温标志" OR "数字量信号"."5区超温标志" OR "数字量信号"."6区超温标志" OR "数字量信号"."7区超温标志" OR "数字量信号"."8区超温标志" OR "数字量信号"."9区超温标志" OR "数字量信号"."10区超温标志" OR "数字量信号"."11区超温标志" OR "数字量信号"."12区超温标志" OR "数字量信号"."13区超温标志" OR "数字量信号"."14区超温标志" OR "数字量信号"."15区超温标志";
END_REGION

REGION Network 18: 消音
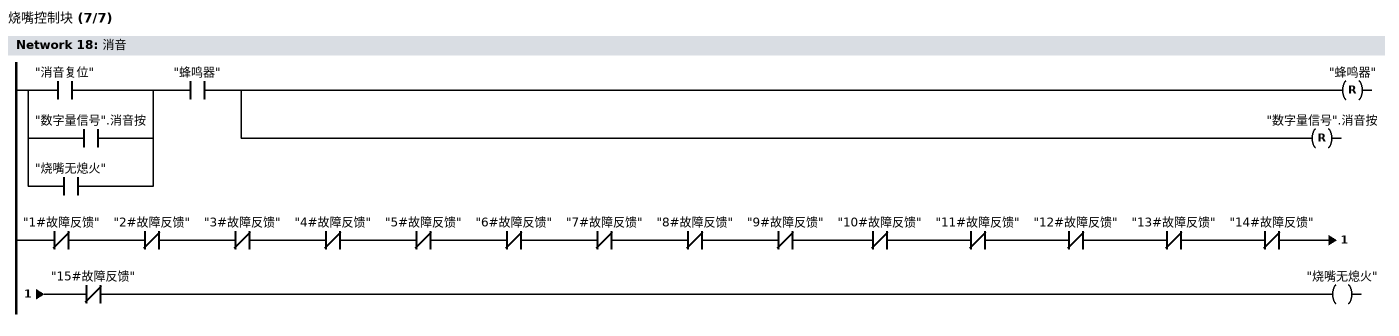
   RUNG wire#powerrail
      Contact( "消音复位" )
      wire#w1
      Contact( "蜂鸣器" )
      wire#w2
      R_Coil( "蜂鸣器" )
   END_RUNG
   RUNG wire#powerrail
      Contact( "数字量信号".消音按 )
   END_RUNG wire#w1
   RUNG wire#powerrail
      Contact( "烧嘴无熄火" )
   END_RUNG wire#w1
   RUNG wire#w2
      R_Coil( "数字量信号".消音按 )
   END_RUNG
   RUNG wire#powerrail
      I_Contact( "1#故障反馈" )
      I_Contact( "2#故障反馈" )
      I_Contact( "3#故障反馈" )
      I_Contact( "4#故障反馈" )
      I_Contact( "5#故障反馈" )
      I_Contact( "6#故障反馈" )
      I_Contact( "7#故障反馈" )
      I_Contact( "8#故障反馈" )
      I_Contact( "9#故障反馈" )
      I_Contact( "10#故障反馈" )
      I_Contact( "11#故障反馈" )
      I_Contact( "12#故障反馈" )
      I_Contact( "13#故障反馈" )
      I_Contact( "14#故障反馈" )
      I_Contact( "15#故障反馈" )
      Coil( "烧嘴无熄火" )
   END_RUNG
   // the same network as SCL:
   #_w1 := ("消音复位" OR "数字量信号".消音按 OR "烧嘴无熄火") AND "蜂鸣器";
   IF #_w1 THEN
       "蜂鸣器" := FALSE;
       "数字量信号".消音按 := FALSE;
   END_IF;
   "烧嘴无熄火" := NOT "1#故障反馈" AND NOT "2#故障反馈" AND NOT "3#故障反馈" AND NOT "4#故障反馈" AND NOT "5#故障反馈" AND NOT "6#故障反馈" AND NOT "7#故障反馈" AND NOT "8#故障反馈" AND NOT "9#故障反馈" AND NOT "10#故障反馈" AND NOT "11#故障反馈" AND NOT "12#故障反馈" AND NOT "13#故障反馈" AND NOT "14#故障反馈" AND NOT "15#故障反馈";
END_REGION
END_FUNCTION
